(*~
		<docu>
			<summary>
				Provides mechanism for delivering static messages to the supervising applications (SCADA/HMI).	
				<remarks>			
					<note type="important">
						Each messenger has a single placeholder for the message; it stores the most important message from the last context cycle. 
						If there are more messages in a single cycle for the same messenger then less important messages are discarded and replaced by 
						the message with the category of higher severity.	
					</note>
				</remarks>			 
			</summary>			
		
		</docu>
~*)
FUNCTION_BLOCK PUBLIC TcoMessenger IMPLEMENTS ITcoMessenger
VAR			
	(*~
		<docu>
			<summary>
				Most important message of this instance of messenger; stores the most important message from the last context cycle. 
				If there are more messages in a single cycle for the same
				messenger then less important messages are discarded and replaced by the message with the category of higher severity.			 
			</summary>			
		</docu>
	~*)
	_mime : TcoMessage;
	_Parent : ITcoObject;
	{attribute clr [ReadOnly()]}
	_contextIdentity : ULINT;	
	{attribute 'hide'}
	_mds : ARRAY[0..MDS_MAX_INDEX] OF TcoMessageDigest;		
END_VAR

VAR CONSTANT
	MDS_MAX_INDEX : INT := 20;
END_VAR

(*~
		<docu>
			<summary>
				Adds message of 'catastrophic' category to the message queue.
				Use this category when there is a situation when the device cannot continue operations due to irrecoverable failure.				 
			</summary>		
		</docu>
~*)
METHOD PUBLIC Catastrophic
VAR_INPUT
	(*~
		<docu>
			<summary>
				Arbitrary message string.			 
			</summary>			
		</docu>
	~*)
	Message : STRING(TcoMessengerSettings.MAX_MESSAGE_TEXT_LENGHT);
END_VAR
THIS^.Post(Message, eMessageCategory.Catastrophic);
END_METHOD

(*~
		<docu>
			<summary>
				Clears the message content.
				<remarks>			
					<note type="important">
						This method is exposed for Rpc calls, for testing purposes. Rpc calls of this method must not be used in production code
					</note>
				</remarks>								 
			</summary>		
		</docu>
~*)
{attribute 'TcRpcEnable'}
METHOD Clear
_mime.TimeStamp :=  DT#1970-01-01-00:00;
_mime.Text := '';
_mime.Identity := 0;
_mime.Category := eMessageCategory.All;
_mime.Cycle := 0;	
_mime.PerCycleCount := 0;
END_METHOD

METHOD PROTECTED Compose : TcoMessage
VAR_INPUT
	Text : STRING(TcoMessengerSettings.MAX_MESSAGE_TEXT_LENGHT);
	Category : eMessageCategory;
END_VAR
IF(_Parent <> 0 AND_THEN _Parent.Context <> 0 AND_THEN _Parent.Context.RealTimeClock <> 0) THEN
	Compose.TimeStamp :=  _Parent.Context.RealTimeClock.NowLocal();	
	Compose.Text := Text;
	Compose.Identity := _Parent.Identity;
	Compose.Category := Category;
	Compose.Cycle := _Parent.Context.StartCycleCount;	
	Compose.MessageDigest := Digest(Text, THIS^._Parent.Context.Environment.Messaging.MessageDigestMethod);
END_IF;
END_METHOD

(*~
		<docu>
			<summary>
				Adds message of 'critical' category to the message queue.
				Use this category when a critical error occured, that is not recoverable by the means of software (reset/restore) and a detailed inspection is required.				 
			</summary>		
		</docu>
~*)
METHOD PUBLIC Critical
VAR_INPUT
	(*~
		<docu>
			<summary>
				Arbitrary message string.			 
			</summary>			
		</docu>
	~*)
	Message : STRING(TcoMessengerSettings.MAX_MESSAGE_TEXT_LENGHT);
END_VAR
THIS^.Post(Message, eMessageCategory.Critical);
END_METHOD

(*~
		<docu>
			<summary>
				Adds message of 'debug' category to the message queue.	
			    Use when you need to report debug information for you as programmer. 			 
			</summary>		
		</docu>
~*)
METHOD PUBLIC Debug
VAR_INPUT
	(*~
		<docu>
			<summary>
				Arbitrary message string.			 
			</summary>			
		</docu>
	~*)
	Message : STRING(TcoMessengerSettings.MAX_MESSAGE_TEXT_LENGHT);
END_VAR
THIS^.Post(Message, eMessageCategory.Debug);
END_METHOD

METHOD Digest : DWORD
VAR_INPUT
	Text : Tc2_System.T_MaxString;
	inDigestType : eMessageDigestMethod;
END_VAR
CASE inDigestType OF
	eMessageDigestMethod.CRC8 :
		Digest := TcoCRC_8(Text);
	eMessageDigestMethod.CRC16 :
		Digest := TcoCRC_16(Text);
	eMessageDigestMethod.CRC32 :
		Digest := TcoCRC_32(Text);
	ELSE
		Digest := 0;
END_CASE
END_METHOD

(*~
		<docu>
			<summary>
				Adds message of 'error' category to the message queue.
				Use this categoty when there is a failure that cannot be immediately recovered and an intervention is needed. This is typically a situation when a device fails
				to deliver expected result. 
				Do not use this category to report information about failed process like measurement or detection.				 
			</summary>						
		</docu>
~*)
METHOD PUBLIC Error
VAR_INPUT
	(*~
		<docu>
			<summary>
				Arbitrary message string.			 
			</summary>			
		</docu>
	~*)
	Message : STRING(TcoMessengerSettings.MAX_MESSAGE_TEXT_LENGHT);
END_VAR
THIS^.Post(Message, eMessageCategory.Error);
END_METHOD

METHOD FB_init : BOOL
VAR_INPUT
	bInitRetains : BOOL; // if TRUE, the retain variables are initialized (warm start / cold start)
	bInCopyCode : BOOL;  // if TRUE, the instance afterwards gets moved into the copy code (online change)
	Parent : ITcoObject;
END_VAR
_Parent := Parent;
_contextIdentity := Parent.Identity;
END_METHOD

(*~
		<docu>
			<summary>
				Adds message of 'information' category to the message queue.	
				Use when you want to deliver information to the user, that has only informative character and does not adversely affect a process.			 
			</summary>			
		</docu>
~*)
METHOD PUBLIC Info 
VAR_INPUT
	(*~
		<docu>
			<summary>
				Arbitrary message string.			 
			</summary>			
		</docu>
	~*)
	Message : STRING(TcoMessengerSettings.MAX_MESSAGE_TEXT_LENGHT);
END_VAR
THIS^.Post(Message, eMessageCategory.Info);
END_METHOD

METHOD PRIVATE LogMessage 
VAR_IN_OUT
	inMessage : TcoMessage;
END_VAR
VAR
	_index : INT;		
END_VAR
CASE _Parent.Context.Environment.Messaging.MessengerLoggingMethod OF
	eMessengerLogMethod.OnEventRisen :
        IF(_Parent.Context.Environment.Messaging.MessageDigestMethod = eMessageDigestMethod.NONE) THEN
			inMessage.MessageDigest := Digest(inMessage.Text, eMessageDigestMethod.CRC8);
		END_IF
			    
		FOR _index := 0 TO MDS_MAX_INDEX DO
			IF(_mds[_index].Cycle = inMessage.Cycle - 1 OR _mds[_index].Cycle = inMessage.Cycle) 
			AND_THEN (_mds[_index].Digest = inMessage.MessageDigest)
			AND_THEN (_mds[_index].Category = inMessage.Category) THEN
			
				IF(inMessage.PerCycleCount <= THIS^.MDS_MAX_INDEX) THEN
					_mds[inMessage.PerCycleCount].Digest := inMessage.MessageDigest;
					_mds[inMessage.PerCycleCount].Cycle := inMessage.Cycle;
					_mds[inMessage.PerCycleCount].Category := inMessage.Category;			
				END_IF;	
				
				RETURN;
				
			END_IF	
		END_FOR
		
		IF(inMessage.PerCycleCount <= THIS^.MDS_MAX_INDEX) THEN
			_mds[inMessage.PerCycleCount].Digest := inMessage.MessageDigest;
			_mds[inMessage.PerCycleCount].Cycle := inMessage.Cycle;
			_mds[inMessage.PerCycleCount].Category := inMessage.Category;
			_Parent.Context.Logger.PushMessage(inMessage);		
		END_IF;
	eMessengerLogMethod.Continuous:
	    _Parent.Context.Logger.PushMessage(inMessage);
END_CASE
END_METHOD

(*~
		<docu>
			<summary>
				Adds message of 'notification' category to the message queue.
				Use this category when you want to report a notification that may be of interest to the user, but does not adveresly affect a process.			 
			</summary>				
		</docu>
~*)
METHOD Notify 
VAR_INPUT
	(*~
		<docu>
			<summary>
				Arbitrary message string.			 
			</summary>			
		</docu>
	~*)
	Message : STRING(TcoMessengerSettings.MAX_MESSAGE_TEXT_LENGHT);
END_VAR
THIS^.Post(Message, eMessageCategory.Notification);
END_METHOD

(*~
		<docu>
			<summary>
				Creates message of given category for this messenger.				 
			</summary>				
		</docu>
~*)
METHOD PUBLIC Post 
VAR_INPUT
	(*~
		<docu>
			<summary>
				Arbitrary message string.			 
			</summary>			
		</docu>
	~*)
	Message : STRING(TcoMessengerSettings.MAX_MESSAGE_TEXT_LENGHT);
	(*~
		<docu>
			<summary>
				Message category.			 
			</summary>			
		</docu>
	~*)
	Category : eMessageCategory;	
END_VAR

VAR
	_wouldBeMime : TcoMessage;
END_VAR
IF(_Parent <> 0 AND_THEN _Parent.Context <> 0 AND_THEN _Parent.Context.Environment <> 0 AND_THEN _Parent.Context.Environment.Messaging <> 0) THEN
	IF(Category < THIS^._Parent.Context.Environment.Messaging.MinLevel
	  OR _Parent.Context.Environment.Messaging.IsSuspended) THEN
		RETURN;
	END_IF; 	
		
	_mime.PerCycleCount := _mime.PerCycleCount + 1;
	_wouldBeMime := Compose(Message, Category);		
	_wouldBeMime.PerCycleCount := _mime.PerCycleCount;
			
    // Same cycle filter for most important messge.
	IF(_mime.Cycle = _Parent.Context.StartCycleCount) THEN		 	
		IF(_wouldBeMime.Category > _mime.Category) THEN	 
			_mime := _wouldBeMime;
		END_IF;
	ELSE
	// Different cycle		
		_wouldBeMime.PerCycleCount := 1;	
		_mime := _wouldBeMime;		
	END_IF;	

	LogMessage(_wouldBeMime);		
END_IF;
END_METHOD

(*~
		<docu>
			<summary>
				Adds message of 'programming error' category to the message queue.	
				Use this category to inform about a possible programming error, defect in settings or missing information at a level of programming or system or process settings.			 
			</summary>				
		</docu>
~*)
METHOD PUBLIC Programming
VAR_INPUT
	(*~
		<docu>
			<summary>
				Arbitrary message string.			 
			</summary>			
		</docu>
	~*)
	Message : STRING(TcoMessengerSettings.MAX_MESSAGE_TEXT_LENGHT);
END_VAR
THIS^.Post(Message, eMessageCategory.ProgrammingError);
END_METHOD

(*~
		<docu>
			<summary>
				Adds message of 'trace' category to the message queue.	
				Use when you need to track detailed information about internal states of the program for detailed visibility. 
				This is lowest level of category that can be used in production, for detailed observation of PLC program.			 
			</summary>					
		</docu>
~*)
METHOD PUBLIC Trace 
VAR_INPUT
	(*~
		<docu>
			<summary>
				Arbitrary message string.			 
			</summary>			
		</docu>
	~*)
	Message : STRING(TcoMessengerSettings.MAX_MESSAGE_TEXT_LENGHT);
END_VAR
THIS^.Post(Message, eMessageCategory.Trace);
END_METHOD

(*~
		<docu>
			<summary>
				Adds message of 'warning' category to the message queue.
				Use this category when you want to report to the user an information about a possible problem, that may adversly affect a process.
				Information in this cateogory aims to help the user to identify a problem, the cause of such problem does not necessarily stops the process.				 
			</summary>					
		</docu>
~*)
METHOD PUBLIC Warning 
VAR_INPUT
	(*~
		<docu>
			<summary>
				Arbitrary message string.			 
			</summary>			
		</docu>
	~*)
	Message : STRING(TcoMessengerSettings.MAX_MESSAGE_TEXT_LENGHT);
END_VAR
THIS^.Post(Message, eMessageCategory.Warning);
END_METHOD

END_FUNCTION_BLOCK

(* stored: Version 1.1.0.1
   POU TcoMessenger: Id {bb89b26f-ec79-4812-bab7-3579b2b6d1be}, SpecialFunc None
   Folder Messages: Id {56442304-2644-4fe1-b5d1-eb5248dd12e5}
   Method Catastrophic: Id {3ead99e7-d4fa-03f6-3060-81990c2076df}
   Method Clear: Id {640fefd4-a9aa-0de1-3f5c-cce4bd50449f}
   Method Compose: Id {3447ad14-6768-48d6-b294-87e00174ef1e}
   Method Critical: Id {a9264967-6c30-0c25-362d-a0380aaea992}
   Method Debug: Id {bd0230f7-b5de-4707-ba4a-f8b17cc23976}
   Method Digest: Id {de6a9eab-3c62-0e43-3529-2cc01fda6c4e}
   Method Error: Id {dc14c403-f11e-4200-ac36-567c3d997bf6}
   Method FB_init: Id {23bbd1ba-9be3-4c0b-a177-bc9de93be447}
   Method Info: Id {d1f4840f-86c5-482b-8fb7-443b9b1c585c}
   Method LogMessage: Id {0b6b2fe7-cb26-02a6-0b72-2570a4f5cb53}
   Method Notify: Id {1595dfe7-5719-459e-bdf2-0e7976c85511}
   Method Post: Id {7e1c7e2b-5612-469e-9139-08754fd973ea}
   Method Programming: Id {1f1b6a21-6158-44a7-b79e-b3fcea42c4e1}
   Method Trace: Id {5a17dee2-c171-4127-9ee1-30d4a06a53bf}
   Method Warning: Id {dd00674c-7475-44d4-8400-894897951e0b} *)
